// TIA Portal V20 export
// export: Created 2025-12-01T14:56:21.3165805Z, ExportSetting None, DisplayName Totally Integrated Automation Portal, DisplayVersion V20 Update 3, DisplayName TIA Portal Openness, DisplayVersion V20 Update 3, DisplayName TIA Portal Version Control Interface, DisplayVersion V20 Update 3, DisplayName STEP 7 Professional, DisplayVersion V20 Update 3, DisplayName STEP 7 Safety, DisplayVersion V20 Update 2, DisplayName WinCC Basic/Comfort/Advanced, DisplayVersion V20 Update 3, DisplayName WinCC Professional, DisplayVersion V20 Update 3, DisplayName WinCC Unified, DisplayVersion V20 Update 3
TYPE "EstadoMaquina_ApiladorDesapilador"
   STRUCT
      Etapa_Reset : Bool;   // Etapa MAQUINA en RESET
      Etapa_EnReposo : Bool;   // Etapa MAQUINA en REPOSO
      Etapa_EnMovimiento : Bool;   // Etapa MAQUINA en MOVIMIENTO
      Etapa_libre_03 : Bool;   // ...
      Etapa_libre_04 : Bool;   // ...
      Etapa_libre_05 : Bool;   // ...
      Etapa_libre_06 : Bool;   // ...
      Etapa_libre_07 : Bool;   // ...
      Etapa_libre_08 : Bool;   // ...
      Etapa_libre_09 : Bool;   // ...
      Etapa_libre_10 : Bool;   // ...
      Etapa_libre_11 : Bool;   // ...
      Etapa_libre_12 : Bool;   // ...
      Etapa_libre_13 : Bool;   // ...
      Etapa_libre_14 : Bool;   // ...
      Manual : Bool;   // MAQUINA EN MANUAL
      Err_Termico_Elevacion : Bool;   // 01. ERROR Termico Elevacion
      Err_Termico_HorquillaDch : Bool;   // 02. ERROR Termico Horquilla Derecha
      Err_Termico_HorquillaIzq : Bool;   // 03. ERROR Termico Horquilla Izquierda
      Err_Posicion : Bool;   // 04. ERROR Posicion
      Byte2_bit4 : Bool;   // 05. ERROR
      Err_TOut_Elevacion : Bool;   // 06. ERROR Timeout Elevacion
      Err_TOut_Recoger_Horquillas : Bool;   // 07. ERROR Timeout Recoger Horquillas
      Err_TOut_Extender_Horquillas : Bool;   // 08. ERROR Timeout Extender Horquillas
      Byte3_bit0 : Bool;   // 09. ERROR
      Byte3_bit1 : Bool;   // 10. ERROR
      Byte3_bit2 : Bool;   // 11. ERROR
      Byte3_bit3 : Bool;   // 12. ERROR
      Byte3_bit4 : Bool;   // 13. ERROR
      Byte3_bit5 : Bool;   // 14. ERROR
      Byte3_bit6 : Bool;   // 15. ERROR
      Byte3_bit7 : Bool;   // 16. ERROR
      Err_Seg_Up : Bool;   // 17. ERROR Micro Seguridad UP
      Err_Seg_Down : Bool;   // 18. ERROR Micro Seguridad DW
      Byte4_bit2 : Bool;   // 19. ERROR
      Byte4_bit3 : Bool;   // 20. ERROR
      Byte4_bit4 : Bool;   // 21. ERROR
      Byte4_bit5 : Bool;   // 22. ERROR
      Byte4_bit6 : Bool;   // 23. ERROR
      Byte4_bit7 : Bool;   // 24. ERROR
      Byte5_bit0 : Bool;   // 25. ERROR
      Byte5_bit1 : Bool;   // 26. ERROR
      Byte5_bit2 : Bool;   // 27. ERROR
      Byte5_bit3 : Bool;   // 28. ERROR
      Byte5_bit4 : Bool;   // 29. ERROR
      Byte5_bit5 : Bool;   // 30. ERROR
      Byte5_bit6 : Bool;   // 31. ERROR
      Byte5_bit7 : Bool;   // 32. ERROR
      Byte6_bit0 : Bool;   // 33. ERROR
      Byte6_bit1 : Bool;   // 34. ERROR
      Byte6_bit2 : Bool;   // 35. ERROR
      Byte6_bit3 : Bool;   // 36. ERROR
      Byte6_bit4 : Bool;   // 37. ERROR
      Byte6_bit5 : Bool;   // 38. ERROR
      Byte6_bit6 : Bool;   // 39. ERROR
      Error_MAQx : Bool;   // Marca General Errol
      En_Termico_Elevacion : Bool;   // Entrada Termico Elevacion
      En_Termico_HorqDch : Bool;   // Entrada Termico Horquilla Derecha
      En_Termico_HorqIzq : Bool;   // Entrada Termico Horquilla Izquierda
      Byte7_bit3 : Bool;   // Entrada 4
      En_ConCarga : Bool;   // Entrada Apilador Con Carga
      En_Lleno : Bool;   // Entrada Status Apilador Lleno
      En_EM_UP : Bool;   // Entrada Detector Final de carrera UP
      En_EM_DW : Bool;   // Entrada Detector Final de carrera DW
      En_PosDOWN : Bool;   // Entrada Apilador Abajo
      En_PosMIDDLE : Bool;   // Entrada Apilador En Pos Media
      En_PosUP : Bool;   // Entrada Apilador Arriba
      Byte8_bit3 : Bool;   // Entrada 12
      En_HorqDrc1_Recogida : Bool;   // ENTRADA Detector Horquilla 1 Derecha Recogida
      En_HorqDrc1_Extendida : Bool;   // ENTRADA Detector Horquilla 1 Derecha Extendida
      En_HorqDrc2_Recogida : Bool;   // ENTRADA Detector Horquilla 2 Derecha Recogida
      En_HorqDrc2_Extendida : Bool;   // ENTRADA Detector Horquilla 2 Derecha Extendida
      En_HorqIzq1_Recogida : Bool;   // ENTRADA Detector Horquilla 1 Izquierda Recogida
      En_HorqIzq1_Extendida : Bool;   // ENTRADA Detector Horquilla 1 Izquierda Extendida
      En_HorqIzq2_Recogida : Bool;   // ENTRADA Detector Horquilla 2 Izquierda Recogida
      En_HorqIzq2_Extendida : Bool;   // ENTRADA Detector Horquilla 2 Izquierda Extendida
      En_Semilleno : Bool;   // Entrada Status Apilador Semilleno
      En_Vacio : Bool;   // Entrada Status Apilador Vacio
      Byte9_bit6 : Bool;   // Entrada 23
      Byte9_bit7 : Bool;   // Entrada 24
      Sa_Subir_Elevacion : Bool;   // Salida SUBIENDO Apilador
      Sa_Bajar_Elevacion : Bool;   // Salida BAJANDO Apilador
      Sa_Recoger_Horquillas : Bool;   // Salida RECOGIENDO Horquillas
      Sa_Extender_Horquillas : Bool;   // Salida EXTENDIENDO Horquillas
      Sa_Extender_HorqDch : Bool;   // Salida EXTENDER HORQUILLA DERECHA
      Sa_Recoger_HorqDch : Bool;   // Salida RECOGER HORQUILLA DERECHA
      Sa_Extender_HorqIzq : Bool;   // SalidaEXTENDER HORQUILLA IZQUIERDA
      Sa_Recoger_HorqIzq : Bool;   // Salida RECOGER HORQUILLA IZQUIERDA
      Byte11_bit0 : Bool;   // Salida 9
      Byte11_bit1 : Bool;   // Salida 10
      Byte11_bit2 : Bool;   // Salida 11
      Byte11_bit3 : Bool;   // Salida 12
      Byte11_bit4 : Bool;   // Salida 13
      Byte11_bit5 : Bool;   // Salida 14
      Byte11_bit6 : Bool;   // Salida 15
      Byte11_bit7 : Bool;   // Salida 16
      Byte12_bit0 : Bool;   // Salida 17
      Byte12_bit1 : Bool;   // Salida 18
      Fin_VI : Bool;   // Fin de Vehiculo
      Paro_Blando : Bool;   // Maquina en paro blando
      Byte12_bit4 : Bool;   // ...
      Byte12_bit5 : Bool;   // ...
      Byte12_bit6 : Bool;   // ...
      Byte12_bit7 : Bool;   // ...
      Byte13_bit0 : Bool;   // ...
      Byte13_bit1 : Bool;   // ...
      Byte13_bit2 : Bool;   // ...
      Byte13_bit3 : Bool;   // ...
      Byte13_bit4 : Bool;   // ...
      Byte13_bit5 : Bool;   // ...
      Byte13_bit6 : Bool;   // ...
      Byte13_bit7 : Bool;   // ...
      Byte14_bit0 : Bool;   // ...
      Byte14_bit1 : Bool;   // ...
      Byte14_bit2 : Bool;   // ...
      Byte14_bit3 : Bool;   // ...
      Byte14_bit4 : Bool;   // ...
      Byte14_bit5 : Bool;   // ...
      Byte14_bit6 : Bool;   // ...
      Byte14_bit7 : Bool;   // ...
      Byte15_bit0 : Bool;   // ...
      Byte15_bit1 : Bool;   // ...
      Byte15_bit2 : Bool;   // ...
      Byte15_bit3 : Bool;   // ...
      Byte15_bit4 : Bool;   // ...
      Byte15_bit5 : Bool;   // ...
      Byte15_bit6 : Bool;   // ...
      Byte15_bit7 : Bool;   // ...
   END_STRUCT;
END_TYPE
